// LS Electric XG5000 project: 66_2_A
// PLC NewPLC
// module base 0 slot 0: 입출력 모듈:XBC-DR20S (DC 24V 입력 12점, 릴레이 출력 8점)

PROGRAM NewProgram (task: 스캔 프로그램)

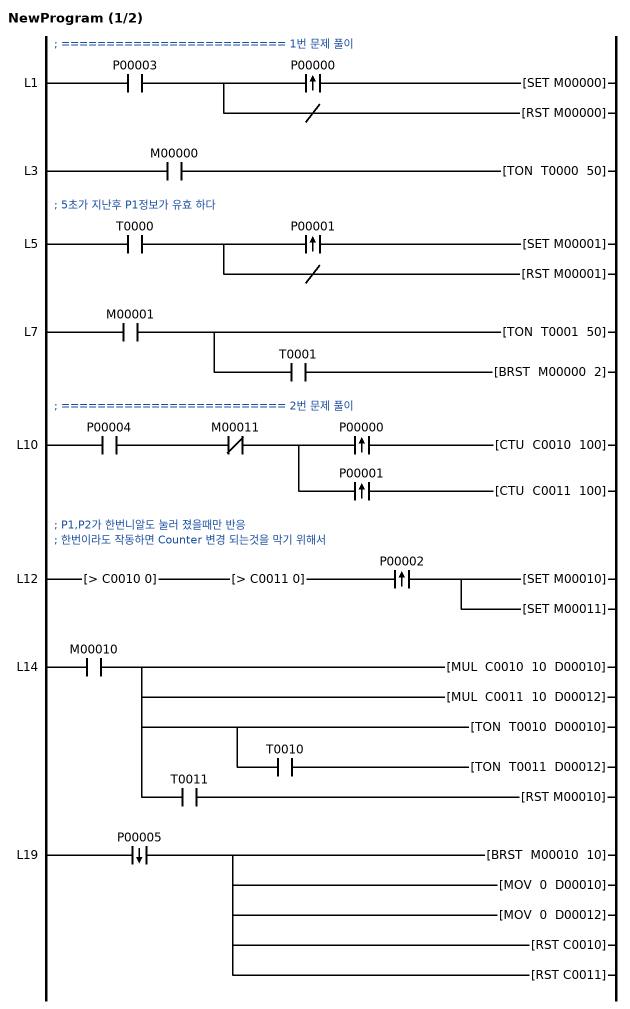
// ========================= 1번 문제 풀이
; L1
LOAD      P00003
MPUSH
ANDP      P00000
SET       M00000
MPOP
NOT
RST       M00000
; L3
LOAD      M00000
TON       T0000 50
; L5
LOAD      T0000
MPUSH
ANDP      P00001
SET       M00001
MPOP
NOT
RST       M00001
// output comment: 5초가 지난후 P1정보가 유효 하다
; L7
LOAD      M00001
TON       T0001 50
AND       T0001
BRST      M00000 2
// ========================= 2번 문제 풀이
; L10
LOAD      P00004
AND NOT   M00011
MPUSH
ANDP      P00000
CTU       C0010 100
MPOP
ANDP      P00001
CTU       C0011 100
; L12
LOAD>     C0010 0
AND>      C0011 0
ANDP      P00002
SET       M00010
SET       M00011
// output comment: P1,P2가 한번니알도 눌러 졌을때만 반응
// output comment: 한번이라도 작동하면 Counter 변경 되는것을 막기 위해서
; L14
LOAD      M00010
MUL       C0010 10 D00010
MUL       C0011 10 D00012
TON       T0010 D00010
MPUSH
AND       T0010
TON       T0011 D00012
MPOP
AND       T0011
RST       M00010
; L19
LOADN     P00005
BRST      M00010 10
MOV       0 D00010
MOV       0 D00012
RST       C0010
RST       C0011

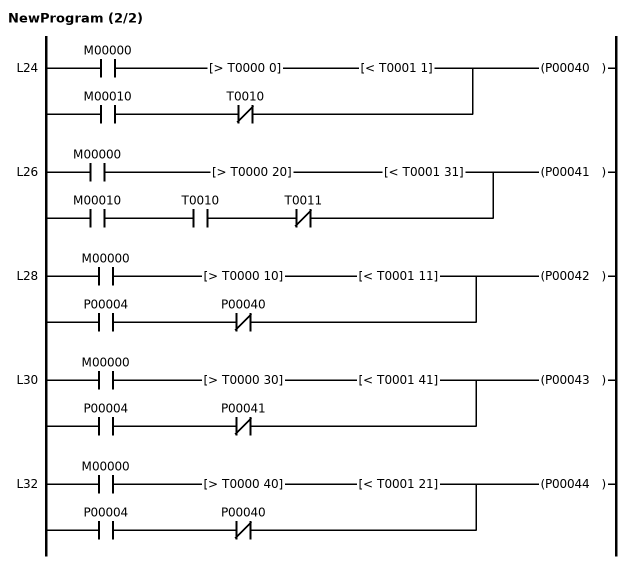
; L24
LOAD      M00000
AND>      T0000 0
AND<      T0001 1
LOAD      M00010
AND NOT   T0010
OR LOAD
OUT       P00040
; L26
LOAD      M00000
AND>      T0000 20
AND<      T0001 31
LOAD      M00010
AND       T0010
AND NOT   T0011
OR LOAD
OUT       P00041
; L28
LOAD      M00000
AND>      T0000 10
AND<      T0001 11
LOAD      P00004
AND NOT   P00040
OR LOAD
OUT       P00042
; L30
LOAD      M00000
AND>      T0000 30
AND<      T0001 41
LOAD      P00004
AND NOT   P00041
OR LOAD
OUT       P00043
; L32
LOAD      M00000
AND>      T0000 40
AND<      T0001 21
LOAD      P00004
AND NOT   P00040
OR LOAD
OUT       P00044